(* PLC project Generated.project, CODESYS CODESYS V3.5 SP19 Patch 1 *)
(* stored: creationDateTime 2026-08-30T23:12:07.033491, modificationDateTime 2026-08-30T23:12:07.033491 *)

(* values of E_ExtractionAssistState: WAIT_BOTTOM_CONFIRMATION: Attente fond Kobold ou attestation opérateur; READY_TO_CLOSE: Prêt à fermer la benne; CLOSING_BUCKET: FB_Bucket ferme M2 seul; CONTROL_ASCENT: M1/M2 synchronisés au palier sans contacteur vitesse; NOMINAL_ASCENT: Ascending couplée avec vitesse demandée opérateur; ERROR_HOLD: Défaut extraction, reprise interdite avant reset *)

{attribute 'qualified_only'}
{attribute 'strict'}
TYPE E_ExtractionAssistState : (WAIT_BOTTOM_CONFIRMATION := 0, READY_TO_CLOSE := 1, CLOSING_BUCKET := 2, CONTROL_ASCENT := 3, NOMINAL_ASCENT := 4, ERROR_HOLD := 5);
END_TYPE

(* values of E_Mode: DISABLE: Mode Désactivé / Veille de sécurité (sorties bloquées); MAINT_N1: Manuel Niveau 1 : Pilotage unitaire avec toutes sécurités actives; MAINT_N2: Manuel Niveau 2 : Pilotage dégradé (droits étendus + bypasses autorisés); SEMI_AUTO: Mode Semi-Automatique (séquenceur automatique) *)

{attribute 'qualified_only'}
{attribute 'strict'}
TYPE E_Mode : (DISABLE := 0, MAINT_N1 := 1, MAINT_N2 := 2, SEMI_AUTO := 3);
END_TYPE

(* ======================================================================= 🧩 ST_Fault — Brique socle défaut (2 vues : live + latchée) ─────────────────────────────────────────────────────────────── 🎯 Rôle : porter l'état défaut d'un composant, applicable dans TOUS les cas (acquittable ou non), sans brique warning séparée. • Vue LIVE (Error / ErrorId) : suit la cause, retombe seule à 0. • Vue LATCHÉE (Latched / LatchedId): mémorisée au défaut, reste jusqu'au front Reset. Le choix acquittable / non-acquittable se fait PAR CAUSE (ST_FaultCause.Latching), jamais par bloc. 🔒 Sécurité : interlock TOUJOURS sur la cause brute (Error / ErrorId), jamais sur l'acquittement. Reset TOUJOURS effectif, jamais conditionné (std §9). 🧬 Composition : brique de base réutilisable — sortie de FB, struct métier, GVL. Texte IHM NON stocké ici : dérivé côté IHM depuis LatchedId / ErrorId. 📄 Doc : DOC/STDS/CODE_QUALITY_STANDARDS.md §2quinquies / §9 ======================================================================= *)
TYPE ST_Fault : STRUCT
  Error : BOOL;  (* <-- [DIAG] vue LIVE : au moins une cause présente maintenant *)
  ErrorId : WORD;  (* <-- [DIAG] bitfield des causes présentes maintenant (0 si aucune) *)
  Latched : BOOL;  (* <-- [DIAG] vue LATCHÉE : défaut non acquitté, reste jusqu'au front Reset *)
  LatchedId : WORD;  (* <-- [DIAG] ErrorId figé à l'apparition du défaut, effacé au Reset *)
END_STRUCT;
END_TYPE

(* ======================================================================= 🧩 ST_FaultCause — Cause élémentaire alimentant ST_Fault (socle FB_FaultCore) ─────────────────────────────────────────────────────────────── 🎯 Rôle : une cause exprimée EN CLAIR (BOOL + libellé), sans bitfield ni masque. Le FB métier remplit une liste (ARRAY[0..15] OF ST_FaultCause) ; le socle FB_FaultCore en déduit ST_Fault (vue live + vue latchée). 🔒 Sécurité : interlock TOUJOURS sur Active (cause brute), jamais sur le latch. Latching = TRUE → la cause ARME la vue latchée (défaut à acquitter). Latching = FALSE → la cause n'alimente que la vue live (retombe seule). Fail-safe : une cause laissée à Latching=FALSE reste visible en live — pour la rendre acquittable, il faut le déclarer explicitement. 📄 Doc : DOC/STDS/CODE_QUALITY_STANDARDS.md §2quinquies / §9 ======================================================================= *)
TYPE ST_FaultCause : STRUCT
  Active : BOOL;  (* 1 = cause présente maintenant (interlock sur cette valeur) *)
  Latching : BOOL;  (* 1 = cause à acquitter (arme Latched) ; 0 = live seulement *)
  Texte : STRING;  (* libellé prêt IHM (non stocké dans ST_Fault, dérivé côté IHM) *)
END_STRUCT;
END_TYPE

(* ======================================================================= 🧩 ST_Lifecycle — Brique socle cycle d'exécution ─────────────────────────────────────────────────────────────── 🎯 Rôle : porter l'avancement d'une action à cycle (organe, séquenceur). Optionnelle : un FB purement synchrone (conditionneur, filtre, joystick) ne la porte pas. 🧬 Composition : brique de base réutilisable, composée avec ST_Fault. 📄 Doc : DOC/STDS/CODE_QUALITY_STANDARDS.md §2quinquies ======================================================================= *)
TYPE ST_Lifecycle : STRUCT
  Busy : BOOL;  (* <-- [STAT] 1 = action en cours *)
  Done : BOOL;  (* <-- [STAT] 1 = action terminée avec succès *)
END_STRUCT;
END_TYPE

(* ======================================================================= ⚙️ FB_ExtractionAssist — Fermeture benne et remontée assistée ─────────────────────────────────────────────────────────────── 🎯 Rôle : Séquence d'extraction (fermeture benne, remontée de contrôle, remontée nominale) 🛡️ Sécurité : Aucune remontée assistée sans fond confirmé, contrôle palier 1 📄 Doc métier : DOC/AF/AF_Partie-04_Mode_SemiAuto_Sequenceur_v2.3.md ======================================================================= *)
FUNCTION_BLOCK FB_ExtractionAssist
  VAR_INPUT
    Enable : BOOL;  (* === COMMANDES & AUTORISATIONS === --> [CMD] Activation generale du FB (TRUE=Autorise) *)
    Reset : BOOL;  (* --> [CMD] Acquittement defaut (front) *)
    PowerContactorEngaged : BOOL;  (* --> [SAFE] Chaine de securite OK *)
    Mode : E_Mode;  (* --> [CMD] Mode de fonctionnement arbitre *)
    MotionRequestActive : BOOL;  (* --> [CMD] Intention de mouvement active *)
    MotionDirection : INT;  (* --> [CMD] Sens de mouvement (+1 = montee) *)
    BottomPositionConfirmed : BOOL;  (* --> [SAFE] Attestation fond confirme (Kobold ou op) *)
    BucketIsClosed : BOOL;  (* === CAPTEURS & ETATS MATERIELS === --> [HW] Benne fermee confirmee *)
    BucketBusy : BOOL;  (* --> [HW] Mouvement benne en cours *)
    BucketError : BOOL;  (* --> [SAFE] Defaut sur sous-systeme benne *)
    WinchSyncError : BOOL;  (* --> [SAFE] Defaut de desynchronisme treuils M1/M2 *)
    M1Position_M : REAL;  (* --> [HW] Position codeur treuil M1 (m) *)
    M2Position_M : REAL;  (* --> [HW] Position codeur treuil M2 (m) *)
    M1MeasuredSpeedValid : BOOL;  (* --> [HW] Validite mesure vitesse M1 *)
    M2MeasuredSpeedValid : BOOL;  (* --> [HW] Validite mesure vitesse M2 *)
    PositionsValid : BOOL;  (* --> [HW] Validite des mesures de position *)
    ControlAscentDistance_M : REAL;  (* === CONFIGURATION & REGLAGES === --> [CFG] Distance palier 1 de controle remontee (m) *)
    CfgBucketCloseTimeout : TIME := TIME#75s0ms;  (* --> [CFG] Backstop fermeture benne (doit rester > BucketMoveTimeout) *)
    BucketMoveTimeout : TIME := TIME#60s0ms;  (* --> [CFG] Reference watchdog mouvement FB_Bucket (verrouillage ordre backstop) *)
    CycleTime : TIME := TIME#10ms;  (* --> [CFG] Base de temps d'integration (periode MainTask) *)
  END_VAR
  VAR_OUTPUT
    Ready : BOOL;  (* === ETATS IEC & DEFECTUOSITES === <-- [STAT] FB pret a fonctionner *)
    Fault : ST_Fault;  (* 🧩 Statut transverse (forme cible ST_Fault + ST_Lifecycle) *)
    Lifecycle : ST_Lifecycle;
    ExtractionState : E_ExtractionAssistState;  (* <-- [STAT] Phase interne extraction *)
    StepAtFault : E_ExtractionAssistState;  (* <-- [DIAG] Phase active memorisee lors du defaut *)
    BucketCloseRequest : BOOL;  (* === ORDRES & AUTORISATIONS === <-- [ACT] Demande de fermeture benne *)
    AscentPermit : BOOL;  (* <-- [ACT] Autorisation de remontee assistee *)
    ExtractionControlActive : BOOL;  (* <-- [ACT] Plafond palier 1 pendant la montee controlee *)
    BottomConfirmationConsumed : BOOL;  (* <-- [STAT] Signal confirmation fond consomme *)
    OperatorActionId : WORD;  (* === DIAGNOSTIC IHM === <-- [DIAG] ID action operateur requise *)
    OperatorAction : STRING(120);  (* <-- [DIAG] Message explicatif operateur *)
  END_VAR
  VAR
    ResetEdge : R_TRIG;  (* === DETECTEURS DE FRONTS === . [LOC] Detecteur front montant Reset *)
    ErrorEdge : R_TRIG;  (* . [LOC] Detecteur front montant apparition defaut *)
    ControlStartM1Position_M : REAL;  (* === MEMORISATIONS & POSITIONS INTERNES === . [LOC] Position M1 au debut du palier de controle (m) *)
    ControlStartM2Position_M : REAL;  (* . [LOC] Position M2 au debut du palier de controle (m) *)
    PrevState : E_ExtractionAssistState;  (* . [LOC] Phase au scan precedent (survit au gate) *)
    CalculatedControlAscentTimeout : TIME;  (* === CALCUL DYNAMIQUE RUNTIME DU TIMEOUT DECOLLAGE === . [LOC] Plafond anti-blocage decollage calcule au runtime *)
    BucketCloseTimerAcc : TIME := TIME#0ms;  (* === ACCUMULATEURS DE TEMPS ANTI-POMPAGE === . [LOC] Temps cumule fermeture benne sous montee demandee *)
    ControlAscentTimerAcc : TIME := TIME#0ms;  (* . [LOC] Temps cumule decollage controle sous montee demandee *)
    ErrorCausePresent : BOOL;  (* === VARIABLES LOCALES INTERNES === . [LOC] Presence d'une cause de defaut parametrage *)
    BucketErrorFault : BOOL;  (* . [LOC] Latch erreur benne *)
    SyncOrSpeedErrorFault : BOOL;  (* . [LOC] Latch erreur synchro/vitesse *)
    TimeoutBucketCloseFault : BOOL;  (* . [LOC] Latch backstop fermeture benne *)
    TimeoutControlAscentFault : BOOL;  (* . [LOC] Latch timeout decollage controle *)
    StepAtFaultCaptured : BOOL;  (* . [LOC] StepAtFault deja fige pour l'episode de defaut courant *)
    AssistPermit : BOOL;  (* . [LOC] Ascending assistee reellement demandee (sens + mode) *)
    AscentControlSafe : BOOL;  (* . [LOC] Entrees [SAFE] saines pour le decollage controle *)
    AscentNominalSafe : BOOL;  (* . [LOC] Entrees [SAFE] saines pour la remontee nominale *)
    CausesPhysiquesEffacees : BOOL;  (* . [LOC] Toutes les entrees defaut treuil/benne revenues a l'etat sain *)
    instFault : FB_FaultCore;  (* === SOCLE DEFAUT === * [INST] Socle défaut transverse *)
    instCauses : ARRAY[0..15] OF ST_FaultCause;  (* . [LOC] Table des causes nommées *)
    CST_MinSpeed_Mps : REAL := 0.15;  (* === CONSTANTES DERIVATION TIMEOUT ANTI-BLOCAGE === Vitesse Palier 1 mini sous charge/mou (m/s) *)
    CST_ControlAscentMargin : REAL := 2;  (* Facteur de marge sur la course de decollage *)
    CST_TimeoutMinDistance_M : REAL := 0.1;  (* Plancher de distance pour le calcul (evite timeout degenere) *)
    CST_TimeoutMaxDistance_M : REAL := 20;  (* Plafond de distance : borne le calcul avant REAL_TO_UDINT (anti-overflow) *)
    CST_BackstopMax : TIME := TIME#600s0ms;  (* Plafond du backstop fermeture benne : au-dela, risque d'overflow de l'accumulateur *)
    CST_SecToMs : REAL := 1000;  (* Conversion secondes -> millisecondes *)
  END_VAR

            

// === IMPLEMENTATION ===

{region "§1 Causes & Socle Défaut (évalué en continu)"}
// 🔑 1. FRONTS
ResetEdge(CLK := Reset);
// Parametrage invalide : distance nulle, backstop nul, base de temps nulle, ou backstop
// qui fauterait AVANT le watchdog benne (masquerait BucketError - ordre des watchdogs).
ErrorCausePresent := (ControlAscentDistance_M <= 0.0)
                  OR (CfgBucketCloseTimeout <= T#0ms)
                  OR (CycleTime <= T#0ms)
                  OR (CfgBucketCloseTimeout <= BucketMoveTimeout)
                  OR (CfgBucketCloseTimeout > CST_BackstopMax);  // borne haute : evite l'overflow de BucketCloseTimerAcc (F3)

// ⏱️ Plafond anti-blocage decollage calcule au runtime : course de controle bornee [plancher..plafond]
// avant conversion REAL->UDINT->TIME (anti-overflow sur valeur IHM aberrante, CQS §6).
CalculatedControlAscentTimeout := UDINT_TO_TIME(REAL_TO_UDINT(
    LIMIT(CST_TimeoutMinDistance_M, ControlAscentDistance_M, CST_TimeoutMaxDistance_M)
    / CST_MinSpeed_Mps * CST_ControlAscentMargin * CST_SecToMs));

// ⏱️ Integrateurs de temps de montee effective (anti-pompage homme-mort)
IF (ExtractionState = E_ExtractionAssistState.CLOSING_BUCKET) AND MotionRequestActive AND (MotionDirection = 1) THEN
    BucketCloseTimerAcc := BucketCloseTimerAcc + CycleTime;
    IF BucketCloseTimerAcc >= CfgBucketCloseTimeout THEN
        TimeoutBucketCloseFault := TRUE;
    END_IF;
END_IF;

IF (ExtractionState = E_ExtractionAssistState.CONTROL_ASCENT) AND MotionRequestActive AND (MotionDirection = 1) THEN
    ControlAscentTimerAcc := ControlAscentTimerAcc + CycleTime;
    IF ControlAscentTimerAcc >= CalculatedControlAscentTimeout THEN
        TimeoutControlAscentFault := TRUE;
    END_IF;
END_IF;

// Etat physique des causes treuil/benne : conditionne l'acquittement des latches a cause persistante (F2).
CausesPhysiquesEffacees := NOT BucketError AND NOT WinchSyncError
                        AND PositionsValid AND M1MeasuredSpeedValid AND M2MeasuredSpeedValid;
IF ResetEdge.Q AND NOT ErrorCausePresent AND NOT MotionRequestActive THEN
    // Latches sans cause physique persistante (timeouts, backstop) : acquittables sur simple front Reset.
    TimeoutBucketCloseFault   := FALSE;
    TimeoutControlAscentFault := FALSE;
    BucketCloseTimerAcc       := T#0ms;
    ControlAscentTimerAcc     := T#0ms;
    StepAtFaultCaptured       := FALSE;
    ExtractionState := E_ExtractionAssistState.WAIT_BOTTOM_CONFIRMATION;
    // Latches de cause physique : acquittables SEULEMENT si l'entree de defaut est revenue saine (F2).
    IF CausesPhysiquesEffacees THEN
        BucketErrorFault      := FALSE;
        SyncOrSpeedErrorFault := FALSE;
    END_IF;
END_IF;

instCauses[1].Active   := BucketErrorFault;
instCauses[1].Latching := TRUE;
instCauses[1].Texte    := 'Defaut sous-systeme benne pendant fermeture';

instCauses[2].Active   := SyncOrSpeedErrorFault;
instCauses[2].Latching := TRUE;
instCauses[2].Texte    := 'Defaut synchro ou capteurs treuils pendant remontee';

instCauses[3].Active   := ErrorCausePresent;
instCauses[3].Latching := TRUE;
instCauses[3].Texte    := 'Parametrage distance de controle ou backstop invalide';

instCauses[4].Active   := TimeoutBucketCloseFault;
instCauses[4].Latching := TRUE;
instCauses[4].Texte    := 'Depassement backstop fermeture benne';

instCauses[5].Active   := TimeoutControlAscentFault;
instCauses[5].Latching := TRUE;
instCauses[5].Texte    := 'Depassement tempo decollage controle';

// Appel du socle de défaut
instFault(Enable := Enable, Reset := Reset, Causes := instCauses);
Fault := instFault.Fault;

// 📸 Capture ordonnee de StepAtFault (D2). Les defauts leves dans le CASE se figent au site du
// latch (voir §3) ; ce bloc ne couvre que les defauts detectes en §1 (backstop, timeout, parametrage),
// ou ExtractionState/PrevState sont encore l'etape reelle. StepAtFaultCaptured evite l'ecrasement.
ErrorEdge(CLK := Fault.Error);
IF ErrorEdge.Q AND NOT StepAtFaultCaptured THEN
    StepAtFault := PrevState;
    StepAtFaultCaptured := TRUE;
ELSIF ResetEdge.Q AND NOT ErrorCausePresent AND NOT MotionRequestActive THEN
    StepAtFault := E_ExtractionAssistState.WAIT_BOTTOM_CONFIRMATION;
END_IF;
{endregion}

{region "§2 Gate neutralisation"}
// 🛑 2. GATE
IF NOT Enable OR NOT PowerContactorEngaged THEN
    Ready := FALSE;
    Lifecycle.Busy := FALSE;
    Lifecycle.Done := FALSE;
    BucketCloseRequest := FALSE;
    AscentPermit := FALSE;
    ExtractionControlActive := FALSE;
    BottomConfirmationConsumed := FALSE;
    ExtractionState := E_ExtractionAssistState.WAIT_BOTTOM_CONFIRMATION;
    // StepAtFault / StepAtFaultCaptured NON reinitialises ici : l'etape figee au defaut reste
    // lisible pour l'IHM/diagnostic apres un cycle Enable OFF->ON ; seul un front Reset l'efface.
    PrevState := E_ExtractionAssistState.WAIT_BOTTOM_CONFIRMATION;
    BucketCloseTimerAcc := T#0ms;
    ControlAscentTimerAcc := T#0ms;
    OperatorActionId := 0;
    OperatorAction := '';
    RETURN;
END_IF;

Ready := Enable AND NOT Fault.Latched;
{endregion}

{region "§3 Machine etat fermeture remontee"}
BucketCloseRequest := FALSE;
AscentPermit := FALSE;
ExtractionControlActive := FALSE;
BottomConfirmationConsumed := FALSE;
Lifecycle.Busy := FALSE;
Lifecycle.Done := FALSE;

// Ascending assistee reellement demandee : sens ascending + mode maintenance (H5, double garde vs Enable PRG_03).
AssistPermit := MotionRequestActive AND (MotionDirection = 1)
            AND (Mode = E_Mode.MAINT_N1 OR Mode = E_Mode.MAINT_N2);
// Entrees [SAFE] saines : coupure meme-scan des permis si defaut treuil/synchro (H2), avant meme le latch.
AscentControlSafe := NOT WinchSyncError AND PositionsValid AND M1MeasuredSpeedValid AND M2MeasuredSpeedValid;
AscentNominalSafe := NOT WinchSyncError AND PositionsValid;

// Garde-fou non-redemarrage auto : un defaut latche non acquitte verrouille la machine
// d'etat en ERROR_HOLD, meme si la vue live Fault.Error retombe (cause disparue).
IF Fault.Error OR Fault.Latched THEN
    ExtractionState := E_ExtractionAssistState.ERROR_HOLD;
    OperatorActionId := 16#0280;
    OperatorAction := 'Vérifier la benne et les treuils puis réarmer avant de reprendre.';
ELSE
    CASE ExtractionState OF
        E_ExtractionAssistState.WAIT_BOTTOM_CONFIRMATION:
            IF BottomPositionConfirmed THEN
                ExtractionState := E_ExtractionAssistState.READY_TO_CLOSE;
            ELSE
                OperatorActionId := 16#0200;
                OperatorAction := 'Confirmer que la benne est posée au fond avant extraction.';
            END_IF;

        E_ExtractionAssistState.READY_TO_CLOSE:
            Ready := TRUE;
            OperatorActionId := 16#0201;
            OperatorAction := 'Demander la montée pour fermer la benne.';
            IF MotionRequestActive AND (MotionDirection = 1) THEN
                BottomConfirmationConsumed := TRUE;
                BucketCloseTimerAcc := T#0ms;   // ⏱️ RAZ a l'entree exacte de CLOSING_BUCKET
                ExtractionState := E_ExtractionAssistState.CLOSING_BUCKET;
            END_IF;

        E_ExtractionAssistState.CLOSING_BUCKET:
            Lifecycle.Busy := TRUE;
            BucketCloseRequest := AssistPermit AND NOT BucketError; // coupure meme-scan sur defaut benne (H2)
            // Autorisation de montee pendant la fermeture : la benne se ferme en montant.
            // Consommee par l'arbitrage (PRG_04) comme permis de montee assistee (H2).
            AscentPermit := AssistPermit AND AscentControlSafe;
            OperatorActionId := 16#0202;
            OperatorAction := 'Maintenir la montée : fermeture de la benne en cours.';
            IF BucketError THEN
                IF NOT StepAtFaultCaptured THEN
                    StepAtFault := ExtractionState;
                    StepAtFaultCaptured := TRUE;
                END_IF;
                BucketErrorFault := TRUE;
            ELSIF BucketIsClosed AND NOT BucketBusy THEN
                ControlStartM1Position_M := M1Position_M;
                ControlStartM2Position_M := M2Position_M;
                ControlAscentTimerAcc := T#0ms;   // ⏱️ RAZ a l'entree exacte de CONTROL_ASCENT
                ExtractionState := E_ExtractionAssistState.CONTROL_ASCENT;
            END_IF;

        E_ExtractionAssistState.CONTROL_ASCENT:
            Lifecycle.Busy := TRUE;
            AscentPermit := AssistPermit AND AscentControlSafe; // coupure meme-scan sur defaut synchro/capteurs (H2)
            ExtractionControlActive := AscentPermit;            // plafond palier 1 suit le permis de montee
            OperatorActionId := 16#0203;
            OperatorAction := 'Maintenir la montée : contrôle charge au palier minimal.';
            IF NOT AscentControlSafe THEN
                IF NOT StepAtFaultCaptured THEN
                    StepAtFault := ExtractionState;
                    StepAtFaultCaptured := TRUE;
                END_IF;
                SyncOrSpeedErrorFault := TRUE;
            ELSIF (M1Position_M >= (ControlStartM1Position_M + ControlAscentDistance_M))
               AND (M2Position_M >= (ControlStartM2Position_M + ControlAscentDistance_M)) THEN
                ExtractionState := E_ExtractionAssistState.NOMINAL_ASCENT;
            END_IF;

        E_ExtractionAssistState.NOMINAL_ASCENT:
            Lifecycle.Busy := TRUE;
            AscentPermit := AssistPermit AND AscentNominalSafe; // coupure meme-scan sur defaut synchro/position (H2)
            OperatorActionId := 16#0204;
            OperatorAction := 'Maintenir la montée : extraction en cours.';
            IF NOT AscentNominalSafe THEN
                IF NOT StepAtFaultCaptured THEN
                    StepAtFault := ExtractionState;
                    StepAtFaultCaptured := TRUE;
                END_IF;
                SyncOrSpeedErrorFault := TRUE;
            END_IF;

        E_ExtractionAssistState.ERROR_HOLD:
            ;
    END_CASE;
END_IF;

// 💾 Memorisation de la phase precedente en toute fin de scan (capture StepAtFault fiable)
PrevState := ExtractionState;
{endregion}

          
END_FUNCTION_BLOCK

(* ======================================================================= 🧩 FB_FaultCore — Socle de remplissage de ST_Fault (vue live + vue latchée) ─────────────────────────────────────────────────────────────── 🎯 Rôle : à partir d'une LISTE de causes en clair (ARRAY[0..15] OF ST_FaultCause), produire la brique ST_Fault : • Error / ErrorId : vue LIVE, suit les causes Active, retombe seule. • Latched / LatchedId: vue LATCHÉE, chaque bit figé à l'apparition d'une cause `Active AND Latching`, conservé jusqu'au front Reset. 🔒 Sécurité : - interlock TOUJOURS sur `Causes[i].Active` (cause brute), jamais sur le latch. - Reset TOUJOURS effectif, jamais conditionné (std §9) — agit même Enable=FALSE. - Latching=FALSE → cause visible en LIVE seulement (fail-safe : reste visible). - un défaut laté non acquitté reste publié même FB désactivé (pas d'effacement silencieux sur bascule Enable OFF→ON sans Reset). - une cause à acquitter réapparue re-arme son bit (ré-alarme). 🧬 Un seul socle, réutilisé par tout FB `standard` qui expose un ST_Fault. Pas de State, pas de Warning, pas de texte — hors périmètre de ce socle. 📄 Doc : DOC/STDS/CODE_QUALITY_STANDARDS.md §2quinquies / §9 ======================================================================= *)
FUNCTION_BLOCK FB_FaultCore
  VAR_INPUT
    Enable : BOOL;  (* --> [CMD] Autorisation générale du FB porteur *)
    Reset : BOOL;  (* --> [CMD] Front d'acquittement (jamais conditionné, §9) *)
    Causes : ARRAY[0..15] OF ST_FaultCause;  (* --> [CMD] Liste des causes en clair (Active / Latching / Texte) *)
  END_VAR
  VAR_OUTPUT
    Ready : BOOL;  (* <-- [STAT] FB porteur autorisé (= Enable) *)
    Fault : ST_Fault;  (* <-- [DIAG] Brique défaut (mappée 1:1 sur la sortie du FB porteur) *)
  END_VAR
  VAR
    ResetEdge : R_TRIG;  (* . [LOC] Front montant Reset *)
    Latch : ARRAY[0..15] OF BOOL;  (* . [LOC] Bit laté par cause, jusqu'au Reset *)
    i : INT;  (* . [LOC] Index de parcours de la liste *)
  END_VAR

            

{region "§1 Reset (front, toujours effectif)"}
// Front Reset : efface tous les latches. Jamais conditionné, agit même Enable=FALSE (§9).
Ready := Enable;
ResetEdge(CLK := Reset);
IF ResetEdge.Q THEN
    FOR i := 0 TO 15 DO Latch[i] := FALSE; END_FOR;
END_IF;
{endregion}

{region "§2 Vue LIVE — Error / ErrorId"}
// Bitfield des causes présentes MAINTENANT. Retombe seule à 0 quand les causes disparaissent.
// Non évaluée si Enable=FALSE (pas de lecture de cause hors autorisation).
Fault.ErrorId := 0;
IF Enable THEN
    FOR i := 0 TO 15 DO
        IF Causes[i].Active THEN
            Fault.ErrorId := Fault.ErrorId OR SHL(WORD#1, INT_TO_DWORD(i));
        END_IF;
    END_FOR;
END_IF;
Fault.Error := (Fault.ErrorId <> 0);
{endregion}

{region "§3 Armement des latches (causes à acquitter)"}
// Une cause Active ET Latching arme son bit ; le bit reste jusqu'au front Reset (§1),
// même si la cause disparaît. Réapparition => ré-armement (ré-alarme).
IF Enable THEN
    FOR i := 0 TO 15 DO
        IF Causes[i].Active AND Causes[i].Latching THEN
            Latch[i] := TRUE;
        END_IF;
    END_FOR;
END_IF;
{endregion}

{region "§4 Vue LATCHÉE — Latched / LatchedId"}
// Toujours publiée, y compris Enable=FALSE : un défaut non acquitté reste visible.
Fault.LatchedId := 0;
FOR i := 0 TO 15 DO
    IF Latch[i] THEN
        Fault.LatchedId := Fault.LatchedId OR SHL(WORD#1, INT_TO_DWORD(i));
    END_IF;
END_FOR;
Fault.Latched := (Fault.LatchedId <> 0);
{endregion}

          
END_FUNCTION_BLOCK
